{attribute 'linkalways'}
{attribute 'hide_all_locals'}
FUNCTION_BLOCK ValueWstring EXTENDS ValueWstringRead IMPLEMENTS Value
VAR
END_VAR

METHOD SetFromType : BOOL
VAR_INPUT
	source : __SYSTEM.AnyType;
END_VAR
SetFromType := ConvertAnyType(source, thisAnyType);
END_METHOD

METHOD SetFromString : BOOL
VAR_INPUT
	value : T_MaxString;
END_VAR
thisValue := STRING_TO_WSTRING(value);

SetFromString := TRUE;
END_METHOD

METHOD Set : BOOL
VAR_INPUT
	source : ANY;
END_VAR
Set := ConvertAnyType(source, thisAnyType);
END_METHOD

END_FUNCTION_BLOCK

(* stored: Version 1.1.0.1
   POU ValueWstring: Id {8a1a00ae-8a07-478d-a0b4-964e0dbbf854}, SpecialFunc None
   Method SetFromType: Id {75a64ec5-171c-44f4-96cd-18c9a9a34153}
   Method SetFromString: Id {9ce71543-d89e-460c-9aea-64fc927676f6}
   Method Set: Id {e31b979f-6617-429e-8006-1c5dbf4784a7} *)
